{attribute 'linkalways'} 
{attribute 'no_explicit_call' := 'This FB is a CLASS and must be accessed using methods or properties'}
{attribute 'enable_dynamic_creation'}
FUNCTION_BLOCK Node_F_VN_OptimalDftSize EXTENDS VisionNode
VAR
    ipImage : _ITcVnImage;
    nOptWidth : _UDINT(0);
    nOptHeight : _UDINT(0);
    hrPrev : _HRESULT(S_OK);
	hresult : _HRESULT(S_OK);
END_VAR

METHOD PUBLIC  Clone : I_Node
VAR
	pNode : POINTER TO Node_F_VN_OptimalDftSize;
END_VAR
pNode := __NEW(Node_F_VN_OptimalDftSize);
Clone := pNode^;
END_METHOD

METHOD FB_init : BOOL
VAR_INPUT
	bInitRetains : BOOL; // if TRUE, the retain variables are initialized (warm start / cold start)
	bInCopyCode : BOOL;  // if TRUE, the instance afterwards gets moved into the copy code (online change)
END_VAR
AddInput('ipImage', ipImage);
AddInput('hrPrev', hrPrev);
AddOutput('nOptWidth', nOptWidth);
AddOutput('nOptHeight', nOptHeight);
AddOutput('hresult',hresult);
END_METHOD

METHOD PROTECTED OnExecute
hresult.Value := F_VN_OptimalDftSize(
    ipImage := ipImage.Value,
	nOptWidth := nOptWidth.Value,
    nOptHeight := nOptHeight.Value,
	hrPrev:= hrPrev.Value);
END_METHOD

METHOD PUBLIC PreExecutionCheck
VAR_INPUT
	Check : I_PreExecutionChecks;
END_VAR
Check.IsTrue(ipImage.IsValid, 'ipImage must contain an image');
END_METHOD

END_FUNCTION_BLOCK

(* stored: Version 1.1.0.1, ProductVersion 3.1.4024.13
   POU Node_F_VN_OptimalDftSize: Id {fdbf95bf-f00e-0f11-33ea-b524a0931e95}, SpecialFunc None
   Folder Constructor: Id {4a3cfd9e-4dc9-0810-3eb0-3344148f2f2d}
   Method Clone: Id {b566351f-fe2f-08a2-2005-0058edd82e36}
   Method FB_init: Id {cfb42660-48b2-0fb8-167e-d3819fdfeccf}
   Method OnExecute: Id {fa93256f-7b78-0dee-0744-a16537696edf}
   Method PreExecutionCheck: Id {7300deec-6181-060f-33bc-c9550290aef6} *)
